Yaskawa INFORM job: FRONT_SEARCH_0ST-2_5240.JBI

/JOB
//NAME FRONT_SEARCH_0ST-2_5240
///FOLDERNAME 02-SKRZYNIE_JOBS
//POS
///NPOS 101,101,0,15,0,0
///TOOL 0
///POSTYPE PULSE
///PULSE
C00000=0,-44333,40442,1,-36510,2
C00001=0,-77502,-19682,2,-20075,2
C00002=-31499,-58302,-23356,15027,12889,-13082
C00003=-52768,-43016,-26078,18373,38595,-18774
C00004=-77982,-19483,-4354,30116,56383,-30765
C00005=-53036,-11528,-12218,12363,64665,-17409
C00006=-53036,-11528,-12218,12363,64665,-17409
C00007=-51536,-9474,-10276,11905,64649,-16876
C00008=-51739,-9114,-7787,12104,63269,-17104
C00009=-53036,-11528,-12218,12363,64665,-17409
C00010=-17541,-26226,-24397,927,59032,-5038
C00011=-17541,-26226,-24397,927,59032,-5038
C00012=-16950,-23991,-22741,715,59568,-4818
C00013=-17036,-23563,-20101,755,58071,-4857
C00014=-17541,-26226,-24397,927,59032,-5038
C00015=34102,-23192,-21614,-15638,64271,13209
C00016=33423,-21885,-20599,-15423,64418,12942
C00017=32426,-19856,-18975,-15106,64629,12551
C00018=32578,-19611,-17013,-15290,63535,12762
C00019=33423,-21885,-20599,-15423,64418,12942
C00020=59339,-6070,-6417,-20979,72191,20891
C00021=59339,-6070,-6417,-20979,72191,20891
C00022=57897,-4256,-4562,-20702,71913,20431
C00023=58108,-3992,-2506,-20878,70835,20713
C00024=59339,-6070,-6417,-20979,72191,20891
C00025=42744,-35904,-30225,-18322,62562,16651
C00026=-53036,-11528,-12218,12363,64665,-17409
C00027=-77982,-26538,-29134,27151,66629,-27745
C00028=-70983,-8594,-1966,26503,59809,-49670
C00029=-80152,19776,40785,37351,72704,-50428
C00030=-79984,20154,42529,37516,71911,-50638
C00031=-79233,18397,40079,37458,71885,-50340
C00032=-79984,20154,42529,37516,71911,-50638
C00033=-73519,23289,38838,28890,77081,-45618
C00034=-73519,24511,42682,29072,75582,-46027
C00035=-73519,23289,38838,28890,77081,-45618
C00036=-88897,15706,42282,50101,71325,-56974
C00037=-88897,15706,42282,50101,71325,-56974
C00038=-87612,12343,37838,50071,70996,-56519
C00039=-85283,14202,40272,50301,69633,-56165
C00040=-87338,12550,38107,50098,70839,-56476
C00041=-84952,-1789,13569,34660,47724,-58955
C00042=-67641,-1674,11109,10330,44856,-44725
C00043=-66443,961,13975,9688,44721,-44210
C00044=-67641,-1674,11109,10330,44856,-44725
C00045=-67641,-376,15347,10694,42950,-44967
C00046=-67641,-1674,11109,10330,44856,-44725
C00047=-79040,417,20398,15965,28992,-57786
C00048=-76655,5212,30978,15501,25024,-57306
C00049=-76655,6949,35816,16758,23084,-57955
C00050=-76655,5212,30978,15501,25024,-57306
C00051=-74761,6919,33010,13466,24593,-56049
C00052=-80460,-2874,12270,15804,32253,-57809
C00053=-61258,-29124,-13156,26560,43617,-22150
C00054=-30420,-40507,-29240,27153,53235,15188
C00055=-18589,-38725,-21450,23338,47896,18931
C00056=-17722,-35233,-16455,23322,46926,19051
C00057=-17722,-33749,-12435,23948,45421,18620
C00058=-17722,-33892,-12819,23887,45564,18661
C00059=-16677,-31133,-11209,23138,46167,19311
C00060=-17819,-35820,-17540,23246,47228,19090
C00061=-74104,-11494,-6266,31916,75042,4269
C00062=-71226,-7329,2631,32115,71468,4273
C00063=-71226,-6504,5446,32343,70365,3922
C00064=-71226,-6611,5086,32313,70505,3967
C00065=-68386,-4058,7675,32040,69573,4789
C00066=-73314,-9412,-353,32206,72648,3829
C00067=51751,-31069,-22965,-10739,49070,48663
C00068=49028,-23852,-11575,-9841,46366,47823
C00069=49028,-23004,-8935,-10039,45204,47956
C00070=49028,-23118,-9286,-10013,45357,47939
C00071=47000,-20813,-7527,-8928,45644,47024
C00072=50476,-26208,-15307,-10408,47325,48332
C00073=90602,-5375,6902,-38786,69848,59444
C00074=83174,19950,50269,-44999,67580,58220
C00075=82362,17902,47383,-44926,67511,57879
C00076=83515,19072,48341,-44798,68200,58056
C00077=78091,19382,40247,-36371,72286,52960
C00078=78091,20664,44011,-36670,70997,53443
C00079=78091,19382,40247,-36371,72286,52960
C00080=88699,7296,38566,-55615,63182,60372
C00081=86803,3068,32674,-55410,62638,59657
C00082=84852,4315,34115,-55564,61561,59330
C00083=86803,3068,32674,-55410,62638,59657
C00084=92770,-2803,21719,-53893,67577,59421
C00085=73393,-10627,10934,-27897,30744,62458
C00086=70789,-6606,18800,-27824,27830,62140
C00087=69654,-4593,20814,-26755,27596,61444
C00088=70789,-6606,18800,-27824,27830,62140
C00089=70789,-5070,23059,-29482,26284,63017
C00090=70789,-6606,18800,-27824,27830,62140
C00091=83486,-8736,6503,-27040,35338,66550
C00092=77831,-2041,26192,-25270,18452,68895
C00093=77967,1961,32070,-26860,17569,69698
C00094=77967,5243,40752,-32914,14549,72656
C00095=77967,1961,32070,-26860,17569,69698
C00096=74560,4730,35257,-21622,16551,66717
C00097=77967,1961,32070,-26860,17569,69698
C00098=81109,-22356,2664,-22493,33121,60116
C00099=86168,-49730,-13668,-23926,46819,49343
C00100=44183,-52048,-7537,-24795,46064,51426
BC00000=887908
BC00001=927819
BC00002=927819
BC00003=927819
BC00004=927819
BC00005=943180
BC00006=943180
BC00007=943180
BC00008=943180
BC00009=943180
BC00010=943180
BC00011=943180
BC00012=943180
BC00013=943180
BC00014=943180
BC00015=943180
BC00016=943180
BC00017=943180
BC00018=943180
BC00019=943180
BC00020=943180
BC00021=943180
BC00022=943180
BC00023=943180
BC00024=943180
BC00025=943180
BC00026=943180
BC00027=943180
BC00028=943180
BC00029=943180
BC00030=943182
BC00031=943182
BC00032=943182
BC00033=943182
BC00034=943182
BC00035=943182
BC00036=943182
BC00037=943182
BC00038=943182
BC00039=943182
BC00040=943182
BC00041=943182
BC00042=943182
BC00043=943182
BC00044=943182
BC00045=943182
BC00046=943182
BC00047=943182
BC00048=943182
BC00049=943182
BC00050=943182
BC00051=943182
BC00052=943182
BC00053=943183
BC00054=943184
BC00055=943184
BC00056=943184
BC00057=943184
BC00058=943184
BC00059=943184
BC00060=943184
BC00061=943184
BC00062=943184
BC00063=943184
BC00064=943184
BC00065=943156
BC00066=943170
BC00067=943170
BC00068=943170
BC00069=943170
BC00070=943170
BC00071=943170
BC00072=943170
BC00073=943184
BC00074=943184
BC00075=943184
BC00076=943184
BC00077=943184
BC00078=943184
BC00079=943184
BC00080=943184
BC00081=943184
BC00082=943184
BC00083=943184
BC00084=943184
BC00085=943184
BC00086=943184
BC00087=943184
BC00088=943184
BC00089=943184
BC00090=943184
BC00091=943184
BC00092=943184
BC00093=943184
BC00094=943184
BC00095=943184
BC00096=943184
BC00097=943184
BC00098=911399
BC00099=884954
BC00100=838173
///POSTYPE BASE
///RECTAN
///RCONF 1,0,0,0,0,0,0,0,0,0,0,0,0,0,0,0,0,0,0,0,0,0,0,0
P00006=0.000,0.000,0.000,0.0000,0.0000,0.0000
///RCONF 0,0,0,0,0,0,0,0,0,0,0,0,0,0,0,0,0,0,0,0,0,0,0,0
P00058=0.000,0.000,3.000,0.0000,0.0000,0.0000
P00350=11.519,-0.008,1.149,0.0000,0.0000,0.0000
P00351=13.563,-0.027,-0.653,0.0000,0.0000,0.0000
P00352=13.252,-0.027,-0.827,0.0000,0.0000,0.0000
P00353=10.971,-0.082,0.776,0.0000,0.0000,0.0000
P00399=-2.449,0.031,8.825,0.0000,0.0000,0.0000
P00400=5.920,-3.503,-0.024,0.0000,0.0000,0.0000
P00401=3.430,-0.021,1.131,0.0000,0.0000,0.0000
P00402=-0.253,1.107,3.062,0.0000,0.0000,0.0000
P00403=-3.666,-0.015,5.328,0.0000,0.0000,0.0000
P00405=2.420,0.007,1.427,0.0000,0.0000,0.0000
P00406=3.513,-0.022,0.429,0.0000,0.0000,0.0000
P00415=-1.781,-1.303,3.250,0.0000,0.0000,0.0000
P00416=0.027,1.119,3.078,0.0000,0.0000,0.0000
//INST
///DATE 2024/06/03 18:55
///ATTR SC,RW
///GROUP1 RB1,BS1
NOP
MOVJ C00000 BC00000 VJ=30.00
MOVJ C00001 BC00001 VJ=20.00
MOVJ C00002 BC00002 VJ=20.00
MOVJ C00003 BC00003 VJ=20.00
MOVJ C00004 BC00004 VJ=10.00
'DODANE
'SZUKANIE FRONT
'------------------------
'503
'------------------------
MOVL C00005 BC00005 V=166.7
MOVL C00006 BC00006 V=66.7 PL=0
REFP 3 C00007 BC00007
CALL JOB:SEARCH-R1
IMOV P0058 V=16.7
SET P0350 P0006
SFTON P0350
REFP 3 C00008 BC00008
CALL JOB:SEARCH-R1
SET P0350 P0006
SFTON P0350
MOVL C00009 BC00009 V=66.7 PL=0
SFTOF
'------------------------
'------------------------
'502
'------------------------
MOVL C00010 BC00010 V=166.7
MOVL C00011 BC00011 V=66.7 PL=0
REFP 3 C00012 BC00012
CALL JOB:SEARCH-R1
IMOV P0058 V=16.7
SET P0351 P0006
SFTON P0351
REFP 3 C00013 BC00013
CALL JOB:SEARCH-R1
SET P0351 P0006
SFTON P0351
MOVL C00014 BC00014 V=66.7 PL=0
SFTOF
'------------------------
'------------------------
'501
'------------------------
MOVL C00015 BC00015 V=166.7
MOVL C00016 BC00016 V=66.7 PL=0
REFP 3 C00017 BC00017
CALL JOB:SEARCH-R1
IMOV P0058 V=16.7
SET P0352 P0006
SFTON P0352
REFP 3 C00018 BC00018
CALL JOB:SEARCH-R1
SET P0352 P0006
SFTON P0352
MOVL C00019 BC00019 V=66.7 PL=0
SFTOF
'------------------------
'------------------------
'500
'------------------------
MOVL C00020 BC00020 V=166.7
MOVL C00021 BC00021 V=66.7 PL=0
REFP 3 C00022 BC00022
CALL JOB:SEARCH-R1
IMOV P0058 V=16.7
SET P0353 P0006
SFTON P0353
REFP 3 C00023 BC00023
CALL JOB:SEARCH-R1
SET P0353 P0006
SFTON P0353
MOVL C00024 BC00024 V=66.7 PL=0
SFTOF
'------------------------
MOVL C00025 BC00025 V=333.3
MOVL C00026 BC00026 V=333.3
MOVJ C00027 BC00027 VJ=10.00
'DODANE
MOVJ C00028 BC00028 VJ=10.00
'------------------------
'SFT402
'------------------------
SFTOF
MOVL C00029 BC00029 V=150.0
MOVL C00030 BC00030 V=66.7 PL=0
REFP 3 C00031 BC00031
CALL JOB:SEARCH-R1
SET P0402 P0006
SFTON P0402
MOVL C00032 BC00032 V=150.0
MOVL C00033 BC00033 V=66.7 PL=0
REFP 3 C00034 BC00034
CALL JOB:SEARCH-R1
SET P0402 P0006
SFTON P0402
MOVL C00035 BC00035 V=133.3
MOVL C00036 BC00036 V=150.0
MOVL C00037 BC00037 V=150.0
MOVL C00038 BC00038 V=66.7 PL=0
REFP 3 C00039 BC00039
CALL JOB:SEARCH-R1
SET P0402 P0006
SFTOF
MOVL C00040 BC00040 V=150.0
'------------------------
'SFT403
'------------------------
'START
SFTOF
MOVL C00041 BC00041 V=250.0
MOVL C00042 BC00042 V=133.3 PL=0
REFP 3 C00043 BC00043
CALL JOB:SEARCH-R1
SET P0416 P0006
SFTON P0416
MOVL C00044 BC00044 V=133.3
REFP 3 C00045 BC00045
CALL JOB:SEARCH-R1
SET P0416 P0006
SFTOF
MOVL C00046 BC00046 V=150.0
'------------------------
'------------------------
SFTOF
MOVL C00047 BC00047 V=250.0
MOVL C00048 BC00048 V=133.3 PL=0
REFP 3 C00049 BC00049
CALL JOB:SEARCH-R1
SET P0403 P0006
SFTON P0403
MOVL C00050 BC00050 V=66.7 PL=0
REFP 3 C00051 BC00051
CALL JOB:SEARCH-R1
SET P0403 P0006
SFTOF
MOVL C00052 BC00052 V=150.0
MOVJ C00053 BC00053 VJ=20.00
MOVJ C00054 BC00054 VJ=20.00
'------------------------
'SFT401
'------------------------
SFTOF
MOVL C00055 BC00055 V=150.0
MOVL C00056 BC00056 V=66.7 PL=0
REFP 3 C00057 BC00057
CALL JOB:SEARCH-R1
SET P0401 P0006
SFTON P0401
MOVL C00058 BC00058 V=66.7 PL=0
REFP 3 C00059 BC00059
CALL JOB:SEARCH-R1
SET P0401 P0006
SFTOF
MOVL C00060 BC00060 V=150.0
'SFT400
'------------------------
SFTOF
MOVL C00061 BC00061 V=333.3
MOVL C00062 BC00062 V=66.7 PL=0
REFP 3 C00063 BC00063
CALL JOB:SEARCH-R1
SET P0405 P0006
SFTON P0405
MOVL C00064 BC00064 V=66.7 PL=0
REFP 3 C00065 BC00065
CALL JOB:SEARCH-R1
SET P0405 P0006
SFTOF
MOVL C00066 BC00066 V=150.0
'SFT400
'------------------------
SFTOF
MOVL C00067 BC00067 V=333.3
MOVL C00068 BC00068 V=133.3 PL=0
REFP 3 C00069 BC00069
CALL JOB:SEARCH-R1
SET P0406 P0006
SFTON P0406
MOVL C00070 BC00070 V=66.7 PL=0
REFP 3 C00071 BC00071
CALL JOB:SEARCH-R1
SET P0406 P0006
SFTOF
MOVL C00072 BC00072 V=150.0
'SFT400
'------------------------
SFTOF
MOVL C00073 BC00073 V=150.0
MOVL C00074 BC00074 V=66.7 PL=0
REFP 3 C00075 BC00075
CALL JOB:SEARCH-R1
SET P0400 P0006
SFTON P0400
MOVL C00076 BC00076 V=150.0
MOVL C00077 BC00077 V=66.7 PL=0
REFP 3 C00078 BC00078
CALL JOB:SEARCH-R1
SET P0400 P0006
SFTON P0400
MOVL C00079 BC00079 V=150.0
MOVL C00080 BC00080 V=150.0
MOVL C00081 BC00081 V=66.7 PL=0
REFP 3 C00082 BC00082
CALL JOB:SEARCH-R1
SET P0400 P0006
SFTOF
MOVL C00083 BC00083 V=83.3
MOVL C00084 BC00084 V=250.0
MOVL C00085 BC00085 V=333.3
MOVL C00086 BC00086 V=66.7 PL=0
REFP 3 C00087 BC00087
CALL JOB:SEARCH-R1
SET P0415 P0006
SFTON P0415
MOVL C00088 BC00088 V=133.3
REFP 3 C00089 BC00089
CALL JOB:SEARCH-R1
SET P0415 P0006
SFTOF
MOVL C00090 BC00090 V=150.0
'------------------------
'SFT403
'------------------------
'START
SFTOF
MOVJ C00091 BC00091 VJ=10.00
'------------------------
'SFT399
'------------------------
'START
SFTOF
MOVL C00092 BC00092 V=150.0
MOVL C00093 BC00093 V=66.7 PL=0
REFP 3 C00094 BC00094
CALL JOB:SEARCH-R1
SET P0399 P0006
SFTON P0399
MOVL C00095 BC00095 V=66.7 PL=0
REFP 3 C00096 BC00096
CALL JOB:SEARCH-R1
SET P0399 P0006
SFTOF
MOVL C00097 BC00097 V=150.0
MOVJ C00098 BC00098 VJ=20.00
MOVJ C00099 BC00099 VJ=30.00
MOVJ C00100 BC00100 VJ=30.00
END
